SUBAPPLICATION mapping_DataPanel (* Subapplication Type *)
  (* Standard: 61499-2 *)
  (* Version 1.0, 2023-01-29, Franz *)
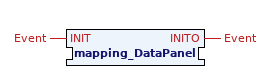
  EVENT_INPUT
    INIT;
  END_EVENT
  EVENT_OUTPUT
    INITO;
  END_EVENT
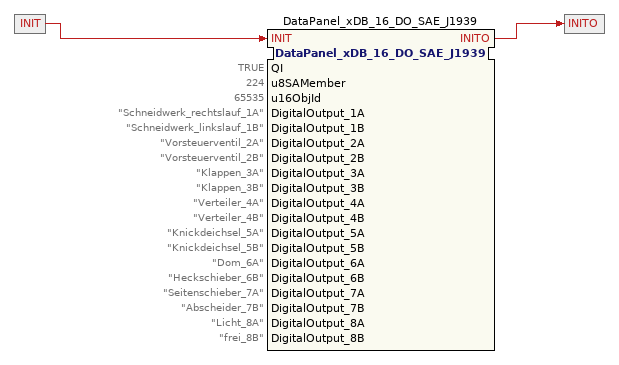
  FBS
    DataPanel_xDB_16_DO_SAE_J1939 : DataPanel_xDB_16_DO_SAE_J1939(QI := TRUE, u8SAMember := 224, u16ObjId := 65535, DigitalOutput_1A := "Schneidwerk_rechtslauf_1A", DigitalOutput_1B := "Schneidwerk_linkslauf_1B", DigitalOutput_2A := "Vorsteuerventil_2A", DigitalOutput_2B := "Vorsteuerventil_2B", DigitalOutput_3A := "Klappen_3A", DigitalOutput_3B := "Klappen_3B", DigitalOutput_4A := "Verteiler_4A", DigitalOutput_4B := "Verteiler_4B", DigitalOutput_5A := "Knickdeichsel_5A", DigitalOutput_5B := "Knickdeichsel_5B", DigitalOutput_6A := "Dom_6A", DigitalOutput_6B := "Heckschieber_6B", DigitalOutput_7A := "Seitenschieber_7A", DigitalOutput_7B := "Abscheider_7B", DigitalOutput_8A := "Licht_8A", DigitalOutput_8B := "frei_8B");
  END_FBS
  EVENT_CONNECTIONS
    INIT TO DataPanel_xDB_16_DO_SAE_J1939.INIT;
    DataPanel_xDB_16_DO_SAE_J1939.INITO TO INITO;
  END_CONNECTIONS
END_SUBAPPLICATION
